FUNCTION_BLOCK FB_Roboter EXTENDS GrundstrukturObjekt
VAR_INPUT
	// Kommunikationsvariablen
	sIP					:T_IPv4Addr;
	iPort				:UINT;
END_VAR

VAR_OUTPUT
END_VAR

VAR
	// Instanziierung von Kommunikationsbausteine
	Connect				:FB_SocketConnect;
	Disconnect			:FB_SocketCloseAll;
	Send				:FB_SocketSend;
	Receive				:FB_SocketReceive;
	
	// Kommunikationsvariablen
	sSrvNetId   		:T_AmsNetId := '';
	tTimeout    		:TIME := T#45S;(*!!!*)
	hSocket    			:T_HSOCKET;
	
	// Managementvariablen
	Connect_State		:BOOL;
	Disconnect_State	:BOOL;
	Switch				:BOOL;
	
	// Testvariable
	test				:BOOL;
	
END_VAR

// Input-Command-Verwaltung
IF iSysCommand = 2 AND iState = 0 THEN			// System schaltet Objekt ein
	Connect_State := TRUE;
END_IF

IF iSysCommand = 1 AND iState = 1 THEN			// System schaltet Objekt aus
	Disconnect_State := TRUE;				
END_IF
//____________________________________________________________________________________________
// Interner Methodenaufruf (Durch System oder Skill)
IF Connect_State THEN
	Switch := Verbinden();
END_IF

IF Disconnect_State THEN
	Switch := Trennen();
END_IF

//____________________________________________________________________________________________
// Zustandsmanagement
CASE iState OF 
	0: // AUS
		// DO
		
		// TRANSITION
			IF Switch THEN							// Verbindung wird aufgebaut
				Connect_State := FALSE;
				Switch := FALSE;
				iState := 1;
			END_IF
			
	//____________________________________________________________________________________________
	1: // BEREIT
		// DO
		
		// TRANSITION
			IF Switch THEN							// Verbindung wird getrennt
				Disconnect_State := FALSE;
				Switch := FALSE;
				iState := 0;
			END_IF
			
			
	
	//____________________________________________________________________________________________
	2: // MANUELL
		// DO
		
		// TRANSITION
	
	//____________________________________________________________________________________________
	3: // LAUFEND
		// DO
		
		// TRANSITION
	
	//____________________________________________________________________________________________
	4: // ABGESCHLOSSEN
		// DO
		
		// TRANSITION
	
	//____________________________________________________________________________________________
	5: // GESTOPPT
		// DO
		
		// TRANSITION
	
	//____________________________________________________________________________________________
	6: // FEHLER
		// DO
		
		// TRANSITION
	
END_CASE

METHOD Trennen : BOOL
VAR_INPUT
END_VAR
// Ausführen von Funktionalitäten
	Disconnect(sSrvNetId := sSrvNetId,
			bExecute := TRUE,
			tTimeout := tTimeout,
			bBusy => bBusy,
			bError => bError,
			nErrId => iErrorID);
	
	IF NOT bBusy AND NOT bError THEN
		Trennen := TRUE;
		Disconnect(bExecute := FALSE);
	END_IF
END_METHOD

METHOD Verbinden : BOOL 
VAR
	
END_VAR
// Ausführen von Funktionalitäten
	Connect(sSrvNetId := sSrvNetId,
			sRemoteHost := sIP,
			nRemotePort := iPort,
			bExecute := TRUE,
			tTimeout := tTimeout,
			bBusy => bBusy,
			bError => bError,
			nErrId => iErrorID,
			hSocket => hSocket);
	
	IF hSocket.handle <> 0 THEN
		Verbinden := TRUE;
		Connect(bExecute := FALSE);
	END_IF
END_METHOD

END_FUNCTION_BLOCK

(* stored: Version 1.1.0.1
   POU FB_Roboter: Id {b3336451-2f79-4a9f-969c-e7cbe82c2874}, SpecialFunc None
   Folder 01_Methoden: Id {1aa946ee-754d-4b9a-827e-c2d8360194ef}
   Folder 01_Nicht-Funktional: Id {dba25a55-927e-456a-8761-8632b877b9de}
   Folder 02_Funktional: Id {c0be9bff-a129-4d21-a449-75936cff3ce2}
   Folder 02_Eigenschaften: Id {678e1a2f-8921-40a4-99a9-2a17bd9f9add}
   Method Trennen: Id {8e6a9714-f7e2-472f-95e7-19c575ef290b}
   Method Verbinden: Id {6eda4363-4e3b-4ff9-8ce0-b02d70060188} *)
